(* IEC 61131-3 sources: volt/packages/volt-lsp-iec/test-corpus/lenze-mid/Device/Plc Logic/Application/Library Manager/(unresolved)/visuusermgmt3 interfaces, 22 files *)

(* ---- VUM_EDITTYPE.dut ---- *)
TYPE VUM_EDITTYPE :
(
	VUM_NONE := 0,
	VUM_ADD := 1,
	VUM_INSERT := 2,
	VUM_MODIFY := 3,
	VUM_REMOVE := 4,
	VUM_CHECKPASSWORD := 5,
	VUM_CHANGEPASSWORD := 6,
	VUM_CHECKPASSWORD_AND_GROUPID := 7,
	VUM_FIND_USER_BY_NAME := 8,
	VUM_FIND_NEXT_ACTIVE_USER_WHICH_BELONGS_TO_ONE_OF_THE_GROUPS := 9
);
END_TYPE

(* ---- VUM_RETURNVALUES.dut ---- *)
TYPE VUM_RETURNVALUES :
(
	ERR_OK := 16#0,
	ERR_FAILED := 16#1,
	ERR_PARAMETER := 16#2,
	ERR_CHANGE_PASSWORD := 16#3F,
	ERR_VUM_FILE_NOT_FOUND := 16#5000,
	ERR_VUM_TEMP_FILE_CANNOT_BE_OPENED := 16#5001,
	ERR_VUM_FILE_READ_FAILED := 16#5002,
	ERR_VUM_FILE_WRITE_FAILED := 16#5003,
	ERR_VUM_INVALID_FILE_CONTENT := 16#5004,
	ERR_VUM_USERNAME_ALREADY_EXIST := 16#5005,
	ERR_VUM_WRONG_PASSWORD := 16#5006,
	ERR_VUM_UNEQUAL_PASSWORD := 16#5007,
	ERR_VUM_NEW_USER_DB_CANNOT_BE_STORED := 16#5008,
	ERR_VUM_ONLY_VISIBLE_USERS_CAN_BE_REMOVED := 16#5009,
	ERR_VUM_EMPTY_PASSWORD_NOT_ALLOWED := 16#500A,
	ERR_VUM_ANOTHER_CLIENT_EDITS_UM := 16#500B,
	ERR_VUM_SYSFILE_ERROR := 16#500C,
	ERR_VUM_SETNEWUSERDB_FAILED := 16#500D,
	ERR_VUM_PROXY_IS_NOT_IN_IDLE_MODE := 16#500E,
	ERR_VUM_DATASERVER_ERROR := 16#500F,
	ERR_VUM_DATASERVER_ERROR_USERS := 16#5010,
	ERR_VUM_MAX_GROUP_LIMIT := 16#5011,
	ERR_VUM_USER_DOES_NOT_EXIST := 16#5012,
	ERR_VUM_USER_IS_INACTIVE := 16#5013,
	ERR_VUM_NO_LOGIN_PROVIDER_AVAILABLE := 16#5014,
	ERR_VUM_NO_CLIENT_MEMORY := 16#5015,
	ERR_VUM_NO_USER_LOGGED_IN := 16#5016,
	ERR_VUM_NO_VALID_USERGROUP_SET := 16#5017,
	ERR_VUM_NO_RIGHT_TO_CHANGE_USERS := 16#5018,
	ERR_VUM_NO_USER_MANAGEMENT := 16#5019,
	ERR_VUM_USER_NOT_IN_USER_GROUP := 16#501A,
	ERR_VUM_EXTERNAL_USER_DATABASE_PROVIDER2_NOT_IMPLEMENTED := 16#501B,
	ERR_VUM_LOGIN_WRONG_ATTEMPT := 16#501C,
	ERR_VUM_LOGIN_SECONDLAST_WRONG_ATTEMPT := 16#501D,
	ERR_VUM_LOGIN_LOCKOUT_TEMP := 16#501E,
	ERR_VUM_LOGIN_LOCKOUT_COMPLETE := 16#501F,
	ERR_VUM_EMPTY_USER_NAME_NOT_ALLOWED := 16#5020,
	ERR_VUM_NOT_ALLOWED_RTS_BASED := 16#5021,
	ERR_VUM_NOT_ALLOWED_LEGACY_BASED := 16#5022,
	ERR_VUM_EQUAL_PASSWORD := 16#5023,
	ERR_VUM_GROUPS_NOT_OK := 16#5024,
	ERR_VUM_NO_ACCESS_RIGHTS := 16#5025
);
END_TYPE

(* ---- VUM_USER.dut ---- *)
TYPE VUM_USER :
STRUCT
	WSTUSERNAME : WSTRING(79);
	WSTFULLNAME : WSTRING(79);
	WSTPASSWORD : WSTRING(79);
	MD5HASH : ARRAY [0..15] OF BYTE;
	DWUSERGROUPID : DWORD;
	ABYUSERGROUPIDS : ARRAY [0..VUM_Constants.VISU_VUM_MAX_GROUPS_PER_USER] OF BYTE;
	BYUSERGROUPCOUNT : BYTE;
	BDEACTIVATED : BOOL;
END_STRUCT
END_TYPE

(* ---- VUM_USER2.dut ---- *)
TYPE VUM_USER2 :
STRUCT
	WSTUSERNAME : WSTRING(79);
	WSTFULLNAME : WSTRING(79);
	DWUSERGROUPID : DWORD;
	ABYUSERGROUPIDS : ARRAY [0..VUM_Constants.VISU_VUM_MAX_GROUPS_PER_USER] OF BYTE;
	BYUSERGROUPCOUNT : BYTE;
	BDEACTIVATED : BOOL;
END_STRUCT
END_TYPE

(* ---- VUM_USER3.dut ---- *)
TYPE VUM_USER3 :
STRUCT
	WSTUSERNAME : WSTRING(79);
	WSTFULLNAME : WSTRING(79);
	WSTPASSWORD : WSTRING(79);
	DWUSERGROUPID : DWORD;
	ABYUSERGROUPIDS : ARRAY [0..VUM_Constants.VISU_VUM_MAX_GROUPS_PER_USER] OF BYTE;
	BYUSERGROUPCOUNT : BYTE;
	BDEACTIVATED : BOOL;
	BCHGPASSFIRSTLOGIN : BOOL;
END_STRUCT
END_TYPE

(* ---- VUM_CONSTANTS.gvl ---- *)
VAR_GLOBAL
	VISU_VUM_MAX_GROUPS_PER_USER : INT := 10;
END_VAR

(* ---- IEXTERNALUSERDATABASEPROVIDER.itf ---- *)
INTERFACE IEXTERNALUSERDATABASEPROVIDER
END_INTERFACE

METHOD CHANGEUSERPASSWORD : VUM_ReturnValues
VAR_INPUT
	WSTUSERNAME : WSTRING;
	WSTNEWPASSWORD : WSTRING;
	WSTOLDPASSWORD : WSTRING;
END_VAR
END_METHOD

METHOD CHECKLOGIN : VUM_ReturnValues
VAR_INPUT
	WSTUSERNAME : WSTRING;
	WSTPASSWORD : WSTRING;
END_VAR
VAR_OUTPUT
	WSTFULLNAME : WSTRING;
	DWUSERGROUPID : DWORD;
END_VAR
END_METHOD

METHOD CHECKLOGINWITHGROUPID : VUM_ReturnValues
VAR_INPUT
	WSTUSERNAME : WSTRING;
	WSTPASSWORD : WSTRING;
	DWUSERGROUPID : DWORD;
END_VAR
VAR_OUTPUT
	WSTFULLNAME : WSTRING;
END_VAR
END_METHOD

METHOD CHANGEUSER : VUM_ReturnValues
VAR_INPUT
	PVUMUSER : POINTER TO VUM_User;
	UDIINDEX : UDINT;
	EEDITTYPE : VUM_EditType;
END_VAR
END_METHOD

METHOD GETUSERCOUNT : UDINT
END_METHOD

METHOD GETUSERS : VUM_ReturnValues
VAR_INPUT
	UDISTARTINDEX : UDINT;
	UDIENDINDEX : UDINT;
	PARR : POINTER TO ARRAY [0..0] OF VUM_User;
	UDIARRSIZE : UDINT;
END_VAR
END_METHOD

(* ---- IEXTERNALUSERDATABASEPROVIDER2.itf ---- *)
INTERFACE IEXTERNALUSERDATABASEPROVIDER2
END_INTERFACE

METHOD FINDUSERBYTYPE : VUM_ReturnValues
VAR_INPUT
	VUMUSERIN : VUM_User;
	EEDITTYPE : VUM_EditType;
END_VAR
VAR_OUTPUT
	VUMUSER : VUM_User;
	UDIINDEX : UDINT;
END_VAR
END_METHOD

(* ---- IVISUUSERMANAGEMENT.itf ---- *)
INTERFACE IVISUUSERMANAGEMENT
END_INTERFACE

METHOD CHECKLOGIN : VUM_ReturnValues
VAR_INPUT
	WSTUSERNAME : WSTRING;
	WSTPASSWORD : WSTRING;
END_VAR
END_METHOD

METHOD CHECKLOGINWITHGROUPID : VUM_ReturnValues
VAR_INPUT
	WSTUSERNAME : WSTRING;
	WSTPASSWORD : WSTRING;
	DWUSERGROUPID : DWORD;
END_VAR
END_METHOD

METHOD REGISTEREXTERNALUSERDATABASEPROVIDER : VUM_ReturnValues
VAR_INPUT
	ITFEXTENALUSERDATABASEPROVIDER : IExternalUserDatabaseProvider;
END_VAR
END_METHOD

(* ---- IVISUUSERMANAGEMENT2.itf ---- *)
INTERFACE IVISUUSERMANAGEMENT2
END_INTERFACE

METHOD LOGINTOUSERGROUP : BOOL
VAR_INPUT
	PCLIENT : POINTER TO BYTE;
	DWGROUPID : DWORD;
	WSTUSERNAME : WSTRING(79);
	WSTFULLNAME : WSTRING(79);
END_VAR
END_METHOD

METHOD LOGINTOUSERGROUPS : BOOL
VAR_INPUT
	PCLIENT : POINTER TO BYTE;
	PADWUSERGROUPIDS : POINTER TO ARRAY [0..0] OF DWORD;
	DWUSERGROUPCOUNT : DWORD;
	WSTUSERNAME : WSTRING(79);
	WSTFULLNAME : WSTRING(79);
END_VAR
END_METHOD

(* ---- IVISUUSERMANAGEMENT3.itf ---- *)
INTERFACE IVISUUSERMANAGEMENT3
END_INTERFACE

METHOD CHANGEPASSWORD : VUM_ReturnValues
VAR_INPUT
	PCLIENT : POINTER TO BYTE;
	WSTUSERNAME : WSTRING(79);
	WSTNEWPASSWORD : WSTRING(79);
	WSTOLDPASSWORD : WSTRING(79);
END_VAR
END_METHOD

METHOD LOGIN : VUM_ReturnValues
VAR_INPUT
	PCLIENT : POINTER TO BYTE;
	WSTUSERNAME : WSTRING(79);
	WSTPASSWORD : WSTRING(79);
END_VAR
VAR_OUTPUT
	WSTFULLNAMEIFAVAILABLE : WSTRING;
	DWUSERGROUPID : DWORD;
	ADWUSERGROUPIDS : ARRAY [0..VUM_Constants.VISU_VUM_MAX_GROUPS_PER_USER] OF DWORD;
	DWUSERGROUPCOUNT : DWORD;
	BDEACTIVATED : BOOL;
END_VAR
END_METHOD

METHOD LOGOUT : VUM_ReturnValues
VAR_INPUT
	PCLIENT : POINTER TO BYTE;
END_VAR
END_METHOD

METHOD USERCOUNT : UDINT
VAR_INPUT
	PCLIENT : POINTER TO BYTE;
END_VAR
VAR_OUTPUT
	RESULT : VUM_ReturnValues;
END_VAR
END_METHOD

METHOD USERS : VUM_ReturnValues
VAR_INPUT
	PCLIENT : POINTER TO BYTE;
	UDISTARTINDEX : UDINT;
	UDIENDINDEX : UDINT;
	PARR : POINTER TO ARRAY [0..0] OF VUM_User2;
	UDIARRSIZE : UDINT;
END_VAR
END_METHOD

(* ---- IVISUUSERMANAGEMENT4.itf ---- *)
INTERFACE IVISUUSERMANAGEMENT4
END_INTERFACE

METHOD EDITUSER : VUM_ReturnValues
VAR_INPUT
	PCLIENT : POINTER TO BYTE;
	PVUMUSERNEW : POINTER TO VUM_User3;
	PVUMUSEROLD : POINTER TO VUM_User3;
	UDIINDEX : UDINT;
	EEDITTYPE : VUM_EditType;
END_VAR
END_METHOD

(* ---- IVISUUSERMGMTCHECKCHANGEUSERREQUESTPARAMETER.itf ---- *)
INTERFACE IVISUUSERMGMTCHECKCHANGEUSERREQUESTPARAMETER
END_INTERFACE

METHOD CHECKCHANGEUSERFLAGS : DWORD
END_METHOD

METHOD CHECKCHANGEUSERINDEX : DWORD
END_METHOD

METHOD CHECKCHANGEUSERTYPE : DWORD
END_METHOD

METHOD GETBUFFER : POINTER TO BYTE
VAR_INPUT
	XSWAPPINGNEEDED : BOOL;
END_VAR
END_METHOD

METHOD GETBUFFERSIZE : UDINT
END_METHOD

(* ---- IVISUUSERMGMTCHECKCHANGEUSERREQUESTRESULT.itf ---- *)
INTERFACE IVISUUSERMGMTCHECKCHANGEUSERREQUESTRESULT
END_INTERFACE

METHOD GETBUFFER : POINTER TO BYTE
END_METHOD

METHOD GETBUFFERSIZE : UDINT
END_METHOD

METHOD SETREADBYTES : BOOL
VAR_INPUT
	UDIREADBYTES : UDINT;
END_VAR
END_METHOD

METHOD SETRESULT
VAR_INPUT
	UDIRESULT : UDINT;
END_VAR
END_METHOD

(* ---- IVISUUSERMGMTCOMMONREQUESTPARAMETER.itf ---- *)
INTERFACE IVISUUSERMGMTCOMMONREQUESTPARAMETER
END_INTERFACE

METHOD GETREQUESTIDENTIFICATION : DataServerRequestIdentification
END_METHOD

METHOD GETREQUESTVERSION : DWORD
END_METHOD

METHOD GETUSERDB : DWORD
END_METHOD

(* ---- IVISUUSERMGMTCOMMONREQUESTRESULT.itf ---- *)
INTERFACE IVISUUSERMGMTCOMMONREQUESTRESULT
END_INTERFACE

METHOD SETERROR
VAR_INPUT
	UDIERROR : UDINT;
END_VAR
END_METHOD

METHOD SETRESULTVERSION
VAR_INPUT
	UDIVERSION : UDINT;
END_VAR
END_METHOD

METHOD SETSWAPPINGNEEDED
VAR_INPUT
	XSWAPPINGNEEDED : BOOL;
END_VAR
END_METHOD

(* ---- IVISUUSERMGMTGETSETDBREQUESTPARAMETER.itf ---- *)
INTERFACE IVISUUSERMGMTGETSETDBREQUESTPARAMETER
END_INTERFACE

METHOD GETSETDBFLAGS : DWORD
END_METHOD

(* ---- IVISUUSERMGMTGETSETDBREQUESTRESULT.itf ---- *)
INTERFACE IVISUUSERMGMTGETSETDBREQUESTRESULT
END_INTERFACE

METHOD SETUSERDB
VAR_INPUT
	UDIUSERDB : UDINT;
END_VAR
END_METHOD

(* ---- IVISUUSERMGMTGETUSERCOUNTREQUESTPARAMETER.itf ---- *)
INTERFACE IVISUUSERMGMTGETUSERCOUNTREQUESTPARAMETER
END_INTERFACE

(* ---- IVISUUSERMGMTGETUSERCOUNTREQUESTRESULT.itf ---- *)
INTERFACE IVISUUSERMGMTGETUSERCOUNTREQUESTRESULT
END_INTERFACE

METHOD SETUSERCOUNT
VAR_INPUT
	UDIUSERCOUNT : UDINT;
END_VAR
END_METHOD

(* ---- IVISUUSERMGMTGETUSERSREQUESTPARAMETER.itf ---- *)
INTERFACE IVISUUSERMGMTGETUSERSREQUESTPARAMETER
END_INTERFACE

METHOD GETENDINDEX : DWORD
END_METHOD

METHOD GETSTARTINDEX : DWORD
END_METHOD

(* ---- IVISUUSERMGMTGETUSERSREQUESTRESULT.itf ---- *)
INTERFACE IVISUUSERMGMTGETUSERSREQUESTRESULT
END_INTERFACE

METHOD GETBUFFER : POINTER TO BYTE
END_METHOD

METHOD GETBUFFERSIZE : UDINT
END_METHOD

METHOD SETREADBYTES : BOOL
VAR_INPUT
	UDIREADBYTES : UDINT;
END_VAR
END_METHOD
